// TIA Portal V20 export
// export: Created 2025-12-01T14:56:11.808816Z, ExportSetting None, DisplayName Totally Integrated Automation Portal, DisplayVersion V20 Update 3, DisplayName TIA Portal Openness, DisplayVersion V20 Update 3, DisplayName TIA Portal Version Control Interface, DisplayVersion V20 Update 3, DisplayName STEP 7 Professional, DisplayVersion V20 Update 3, DisplayName STEP 7 Safety, DisplayVersion V20 Update 2, DisplayName WinCC Basic/Comfort/Advanced, DisplayVersion V20 Update 3, DisplayName WinCC Professional, DisplayVersion V20 Update 3, DisplayName WinCC Unified, DisplayVersion V20 Update 3
TYPE "UDT_Accesos"
   STRUCT
      Memorias : Struct
         MPeticion : Bool;
         MPermiso : Bool;
         MEntradaPeticion : Bool;
         Libre_03 : Bool;
         Libre_04 : Bool;
         Libre_05 : Bool;
         TodasMesas_EnParo : Bool;
         AlgunaMesa_EnMarcha : Bool;
         MFP_ParoBlando : Bool;
         MFP_Marcha : Bool;
         MFP_PulsadorPeticion : Bool;
         Libre_13 : Bool;
         Libre_14 : Bool;
         Libre_15 : Bool;
         Libre_16 : Bool;
         Libre_17 : Bool;
      END_STRUCT;
      Mesas : Array[1..20] of UInt;
   END_STRUCT;
END_TYPE
